FUNCTION_BLOCK FB_AutomaticControl_old
VAR_INPUT
	bEnable								: BOOL;
	bStartMotion 						: BOOL;
	bStopMotion 						: BOOL;
	stValveOutputGeneratorSettings  	: ST_ValveOutputGeneratorSettings;
	stParam 		: ST_Parameters; 
END_VAR
VAR_OUTPUT
	fTime : LREAL;
	fNormalizedValveOpeningRefSignal : LREAL;
END_VAR
VAR
	fbClock 					: FB_Clock;	
	fbValveOutputGenerator 		: FB_ValveOutputGenerator;	
END_VAR

fbClock(
	bEnable := bEnable,
	bStart := bStartMotion,
	bStop := bStopMotion,
	fCycleTime := stParam.fCyclicTime
);

fbValveOutputGenerator(
	bEnable := bEnable,
	stValveOutputGeneratorSettings := stValveOutputGeneratorSettings,
	fClock_s := fbClock.fTime
);

fNormalizedValveOpeningRefSignal := fbValveOutputGenerator.fNormalizedValveOutputRef;
fTime := fbClock.fTime;

END_FUNCTION_BLOCK

(* stored: Version 1.1.0.1, ProductVersion 3.1.4024.11
   POU FB_AutomaticControl_old: Id {b543be1d-46f1-4ea5-ae35-9d7ea7728984}, SpecialFunc None *)
